FUNCTION_BLOCK Jack2Ctrl (* Basic Function Block Type *)
  (* Standard: 61499-2 *)
  (* Version 0.0, 3/23/2016, Aalto_IT, nxtControl GmbH, Template *)
  PACKAGE Main;
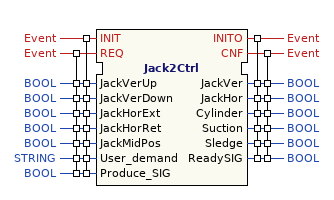
  EVENT_INPUT
    INIT WITH JackVerUp, JackVerDown, JackHorExt, JackHorRet, JackMidPos, User_demand, Produce_SIG; (* Initialization Request *)
    REQ WITH JackVerUp, JackVerDown, JackHorExt, JackHorRet, JackMidPos, User_demand, Produce_SIG; (* Normal Execution Request *)
  END_EVENT
  EVENT_OUTPUT
    INITO WITH JackVer, JackHor, Cylinder, Suction, Sledge, ReadySIG; (* Initialization Confirm *)
    CNF WITH JackVer, JackHor, Cylinder, Suction, Sledge, ReadySIG; (* Execution Confirmation *)
  END_EVENT
  VAR_INPUT
    JackVerUp : BOOL;
    JackVerDown : BOOL;
    JackHorExt : BOOL;
    JackHorRet : BOOL;
    JackMidPos : BOOL;
    User_demand : STRING;
    Produce_SIG : BOOL;
  END_VAR
  VAR_OUTPUT
    JackVer : BOOL;
    JackHor : BOOL;
    Cylinder : BOOL;
    Suction : BOOL;
    Sledge : BOOL;
    ReadySIG : BOOL;
  END_VAR
  VAR
    TimeStamp : DATE_AND_TIME;
  END_VAR
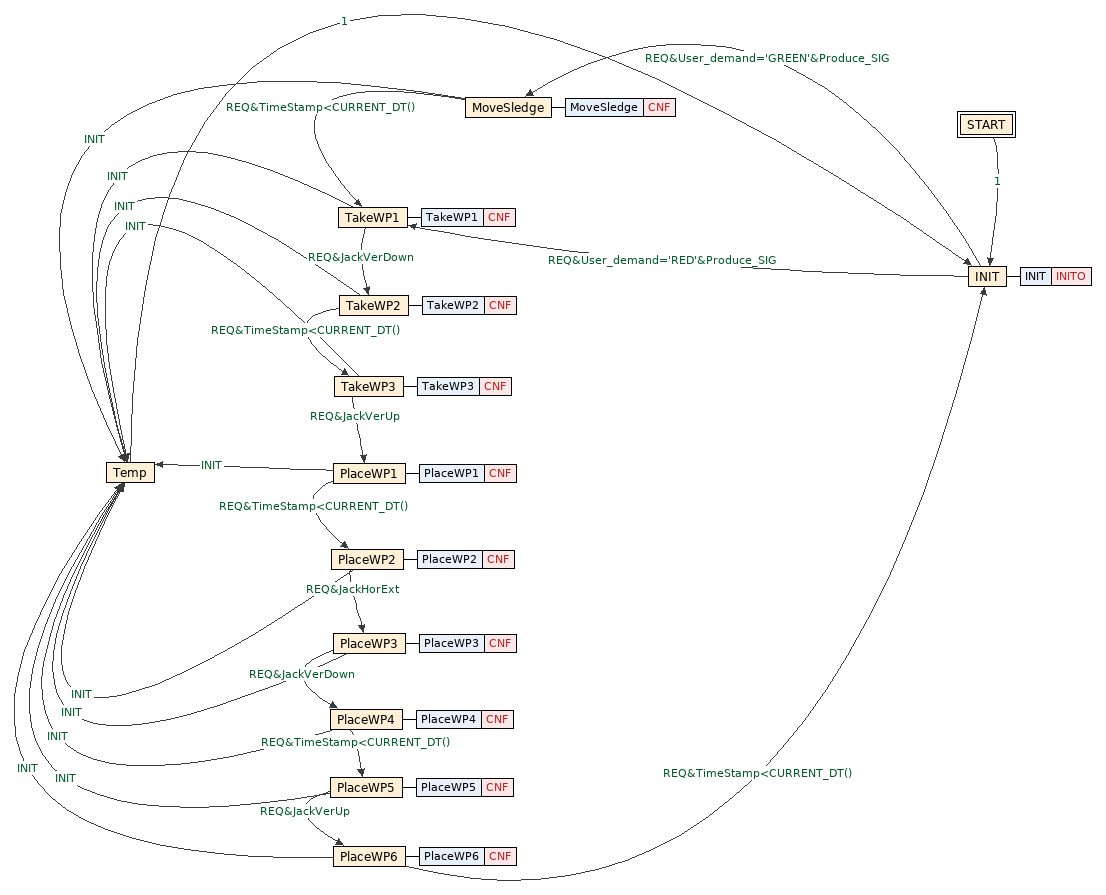
  EC_STATES
    START; (* Initial State *)
    INIT : INIT -> INITO; (* Initialization *)
    Temp;
    MoveSledge : MoveSledge -> CNF;
    TakeWP1 : TakeWP1 -> CNF;
    TakeWP2 : TakeWP2 -> CNF;
    TakeWP3 : TakeWP3 -> CNF;
    PlaceWP1 : PlaceWP1 -> CNF;
    PlaceWP2 : PlaceWP2 -> CNF;
    PlaceWP3 : PlaceWP3 -> CNF;
    PlaceWP4 : PlaceWP4 -> CNF;
    PlaceWP5 : PlaceWP5 -> CNF;
    PlaceWP6 : PlaceWP6 -> CNF;
  END_STATES
  EC_TRANSITIONS
    Temp TO INIT := 1;
    START TO INIT := 1;
    MoveSledge TO TakeWP1 := REQ&TimeStamp<CURRENT_DT();
    TakeWP1 TO TakeWP2 := REQ&JackVerDown;
    TakeWP2 TO TakeWP3 := REQ&TimeStamp<CURRENT_DT();
    TakeWP3 TO PlaceWP1 := REQ&JackVerUp;
    PlaceWP1 TO PlaceWP2 := REQ&TimeStamp<CURRENT_DT();
    PlaceWP2 TO PlaceWP3 := REQ&JackHorExt;
    PlaceWP3 TO PlaceWP4 := REQ&JackVerDown;
    PlaceWP4 TO PlaceWP5 := REQ&TimeStamp<CURRENT_DT();
    PlaceWP5 TO PlaceWP6 := REQ&JackVerUp;
    PlaceWP6 TO Temp := INIT;
    PlaceWP5 TO Temp := INIT;
    PlaceWP4 TO Temp := INIT;
    PlaceWP3 TO Temp := INIT;
    PlaceWP2 TO Temp := INIT;
    MoveSledge TO Temp := INIT;
    TakeWP1 TO Temp := INIT;
    TakeWP2 TO Temp := INIT;
    TakeWP3 TO Temp := INIT;
    PlaceWP1 TO Temp := INIT;
    INIT TO MoveSledge := REQ&User_demand='GREEN'&Produce_SIG;
    INIT TO TakeWP1 := REQ&User_demand='RED'&Produce_SIG;
    PlaceWP6 TO INIT := REQ&TimeStamp<CURRENT_DT();
  END_TRANSITIONS
  ALGORITHM INIT IN ST: (* Initialization algorithm *)
JackVer:=0;
JackHor:=0;
Cylinder:=0;
Suction:=0;
Sledge:=0;
ReadySIG:=0;
  END_ALGORITHM
  ALGORITHM MoveSledge IN ST:
;
JackVer:=0;
JackHor:=0;
Cylinder:=0;
Suction:=0;
Sledge:=0;
ReadySIG:=0;
Sledge:=1; // Move Sledge to second position...
TimeStamp := ADD_DT_TIME(CURRENT_DT(),T#0.3s);
  END_ALGORITHM
  ALGORITHM TakeWP1 IN ST:
;
// Bring the Jack Nose down.
JackVer:=1; // go down.
JackHor:=0;
Cylinder:=0;
Suction:=0;
//Sledge:=0;
ReadySIG:=0;
  END_ALGORITHM
  ALGORITHM TakeWP2 IN ST:
;
// Suction ON and exit after time out.
JackVer:=1;
JackHor:=0;
Cylinder:=0;
Suction:=1; // Suction ON.
//Sledge:=0;
ReadySIG:=0;
TimeStamp := ADD_DT_TIME(CURRENT_DT(),T#0.2s);
  END_ALGORITHM
  ALGORITHM TakeWP3 IN ST:
;
// Go Back UP.
JackVer:=0; // go up with wp.
JackHor:=0;
Cylinder:=0;
Suction:=1;
//Sledge:=0;
ReadySIG:=0;
  END_ALGORITHM
  ALGORITHM PlaceWP1 IN ST:
;
// Bring Sledge back to orig pos if it was moved.
JackVer:=0;
JackHor:=0;
Cylinder:=0;
Suction:=1; // Suction remains ON.
Sledge :=0; // bring sledge back to original pos.
ReadySIG:=0;
TimeStamp := ADD_DT_TIME(CURRENT_DT(),T#0.2s);
  END_ALGORITHM
  ALGORITHM PlaceWP2 IN ST:
;
// Extend the Jack.
JackVer:=0;
JackHor:=1;
Cylinder:=0;
Suction:=1; // remains on.
Sledge:=0;
ReadySIG:=0;
  END_ALGORITHM
  ALGORITHM PlaceWP3 IN ST:
;
// Lower the Nose while extending.
JackVer:=1; // Lower.
JackHor:=1;
Cylinder:=0;
Suction:=1; // remains on.
Sledge:=0;
ReadySIG:=0;
  END_ALGORITHM
  ALGORITHM PlaceWP4 IN ST:
;
// Shut off the Suction.
JackVer:=1; // Lower.
JackHor:=1;
Cylinder:=0;
Suction:=0;
Sledge:=0;
ReadySIG:=0;
TimeStamp := ADD_DT_TIME(CURRENT_DT(),T#0.2s);
  END_ALGORITHM
  ALGORITHM PlaceWP5 IN ST:
;
// Unlower the Jack...
JackVer:=0; // Un-Lower the Jack.
JackHor:=1;
Cylinder:=0;
Suction:=0;
Sledge:=0;
ReadySIG:=0;
  END_ALGORITHM
  ALGORITHM PlaceWP6 IN ST:
;
// Put it back to original position...
JackVer:=0;
JackHor:=0; // Put it back...
Cylinder:=0;
Suction:=0;
Sledge:=0;
ReadySIG:=1; // we are done.
TimeStamp := ADD_DT_TIME(CURRENT_DT(),T#1.0s);
  END_ALGORITHM
END_FUNCTION_BLOCK
